{attribute 'linkalways'} 
{attribute 'no_explicit_call' := 'This FB is a CLASS and must be accessed using methods or properties'}
{attribute 'enable_dynamic_creation'}
FUNCTION_BLOCK Node_F_VN_FillContainerExp_TcVnRectangle_DINT EXTENDS VisionNode
VAR
    ipContainer : _ITcVnContainer;
    stValue : _TcVnRectangle_DINT;
    nStartIdx : _ULINT(0);
    nCount : _ULINT(0);
    hrPrev : _HRESULT(S_OK);
    hresult : _HRESULT(S_OK);
END_VAR

METHOD PUBLIC  Clone : I_Node
VAR
    pNode : POINTER TO Node_F_VN_FillContainerExp_TcVnRectangle_DINT;
END_VAR
pNode := __NEW(Node_F_VN_FillContainerExp_TcVnRectangle_DINT);
Clone := pNode^;
END_METHOD

METHOD FB_init : BOOL
VAR_INPUT
    bInitRetains : BOOL; // if TRUE, the retain variables are initialized (warm start / cold start)
    bInCopyCode : BOOL;  // if TRUE, the instance afterwards gets moved into the copy code (online change)
END_VAR
AddInput('ipContainer', ipContainer);
AddInput('stValue', stValue);
AddParameter('nStartIdx', nStartIdx);
AddParameter('nCount', nCount);
AddInput('hrPrev', hrPrev);
AddOutput('ipContainer', ipContainer);
AddOutput('hresult',hresult);
END_METHOD

METHOD PROTECTED OnExecute
hresult.Value := F_VN_FillContainerExp_TcVnRectangle_DINT(
    ipContainer := ipContainer.Value,
    stValue := stValue.Value,
    nStartIdx := nStartIdx.Value,
    nCount := nCount.Value,
    hrPrev:= hrPrev.Value);
END_METHOD

METHOD PUBLIC PreExecutionCheck
VAR_INPUT
    Check : I_PreExecutionChecks;
END_VAR
Check.IsTrue(ipContainer.IsValid, 'ipContainer must be a valid container');
Check.IsTrue(ipContainer.IsType(TC_GLOBAL_CONST_LIST.ContainerType_Vector_TcVnRectangle_DINT), 'ipContainer contains incorrect type');
END_METHOD

END_FUNCTION_BLOCK

(* stored: Version 1.1.0.1, ProductVersion 3.1.4026.13
   POU Node_F_VN_FillContainerExp_TcVnRectangle_DINT: Id {61083804-5b19-4ddf-841f-9e8db67de85f}, SpecialFunc None
   Folder Constructor: Id {5c6ae3b9-b2b6-425e-9764-1d59657203f8}
   Method Clone: Id {5c464e67-a702-473c-b868-e38e2458bd48}
   Method FB_init: Id {3e320463-cab0-43ac-8bd2-b6d11560db1d}
   Method OnExecute: Id {570e609d-ee31-4e45-afd2-c939c1a8ba6d}
   Method PreExecutionCheck: Id {b7ac60f8-7b1a-453f-8490-6b2e2fae55f4} *)
